RoboDK station: ClassTest.rdk

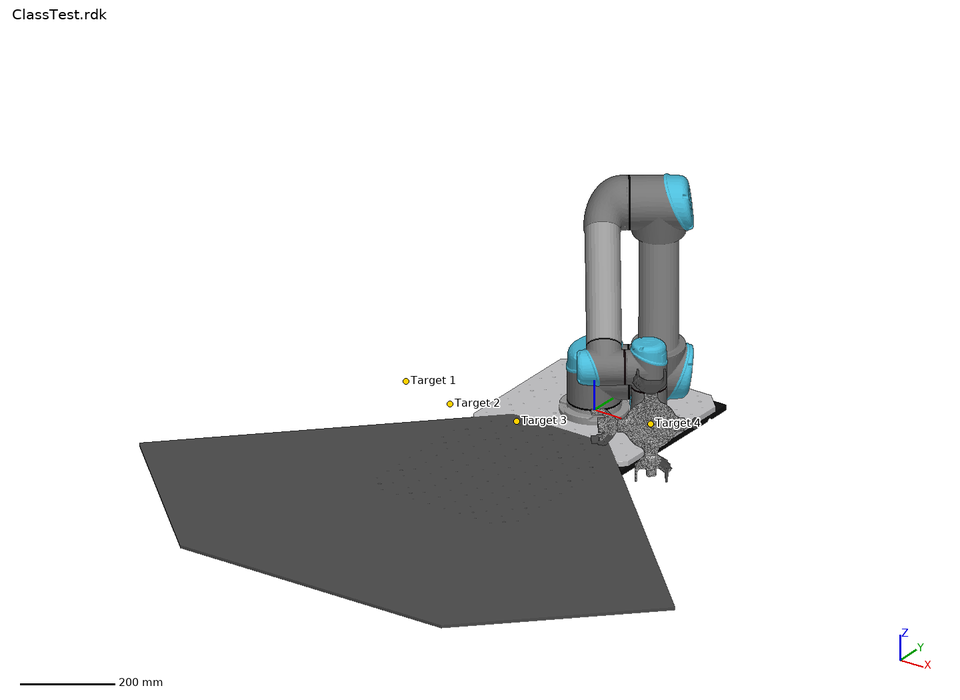
[picture v0: the station drawn from its stored meshes, robots at their saved joint values, targets as dots, program paths as lines]
Station P2 - Robot Cell (saved by RoboDK 5.5.3). Poses are relative to the parent item; angles as X-Y-Z fixed-axis rotations.
Station parameters (name, value as stored): IO_0, 0, IO_1, 1, 10, 0, 11, 0, 12, 1
  - frame UR5 Base at (0, 0, 0) mm
    - robot UR5: 6 axes
        modified DH rows (alpha deg, a mm, theta deg, d mm): 0, 0, 0, 89.2; 90, 0, 180, 0; 0, 425, 0, 0; 0, 392, 0, 109.3; -90, 0, 0, 94.75; 90, 0, 0, 82.5
        joint limits [-360, -360, -360, -360, -360, -360] to [360, 360, 360, 360, 360, 360]; home [0, -90, -90, 0, 90, 0]; saved at [125.87, -83.08, 119.4, -38.13, 88.09, -180]
      - tool GripperAssembled, TCP at (0, 0, 0) mm, size 226.2 x 248.1 x 43.3 mm, geometry from GripperAssembled.step
    - object RobotCellTable at (0, 0, 0) mm, rotated rx 0 ry 0 rz 180 deg, size 1378.2 x 1242.6 x 30 mm, geometry from RobotCellTable.step
    - target Target 1 (joint target) at (-183.8, -428.35, 186.83) mm, rotated rx 2.21 ry -88.19 rz 52.55 deg; joints [52.87, -83.08, 119.4, -38.13, 88.11, 89.99] of UR5
    - target Target 2 (joint target) at (-45.52, -463.89, 186.83) mm, rotated rx 88.19 ry 0.06 rz -17.62 deg; joints [70.49, -83.08, 119.4, -38.13, 88.11, 0] of UR5
    - target Target 3 (joint target) at (116.99, -451.2, 186.83) mm, rotated rx -1.89 ry 88.19 rz -89.37 deg; joints [90.63, -83.08, 119.4, -38.13, 88.11, -90] of UR5
    - target Target 4 (joint target) at (355.89, -301.01, 186.83) mm, rotated rx -88.19 ry -0.06 rz -142.24 deg; joints [125.87, -83.08, 119.4, -38.13, 88.11, -180] of UR5
    - target T5 (joint target) at (-183.78, -428.36, 186.83) mm, rotated rx -88.19 ry -0.06 rz 144.78 deg; joints [52.87, -83.08, 119.4, -38.13, 88.09, -180] of UR5
    - target T6 (joint target) at (-183.78, -428.36, 186.83) mm, rotated rx -88.19 ry -0.06 rz 144.78 deg; joints [54.36, -83.08, 119.4, -38.13, 88.09, -180] of UR5
    - target T7 (joint target) at (-183.78, -428.36, 186.83) mm, rotated rx -88.19 ry -0.06 rz 144.78 deg; joints [55.85, -83.08, 119.4, -38.13, 88.09, -180] of UR5
    - target T8 (joint target) at (-183.78, -428.36, 186.83) mm, rotated rx -88.19 ry -0.06 rz 144.78 deg; joints [57.339, -83.08, 119.4, -38.13, 88.09, -180] of UR5
    - target T9 (joint target) at (-183.78, -428.36, 186.83) mm, rotated rx -88.19 ry -0.06 rz 144.78 deg; joints [58.829, -83.08, 119.4, -38.13, 88.09, -180] of UR5
    - target T10 (joint target) at (-183.78, -428.36, 186.83) mm, rotated rx -88.19 ry -0.06 rz 144.78 deg; joints [60.319, -83.08, 119.4, -38.13, 88.09, -180] of UR5
    - target T11 (joint target) at (-183.78, -428.36, 186.83) mm, rotated rx -88.19 ry -0.06 rz 144.78 deg; joints [61.809, -83.08, 119.4, -38.13, 88.09, -180] of UR5
    - target T12 (joint target) at (-183.78, -428.36, 186.83) mm, rotated rx -88.19 ry -0.06 rz 144.78 deg; joints [63.299, -83.08, 119.4, -38.13, 88.09, -180] of UR5
    - target T13 (joint target) at (-183.78, -428.36, 186.83) mm, rotated rx -88.19 ry -0.06 rz 144.78 deg; joints [64.788, -83.08, 119.4, -38.13, 88.09, -180] of UR5
    - target T14 (joint target) at (-183.78, -428.36, 186.83) mm, rotated rx -88.19 ry -0.06 rz 144.78 deg; joints [66.278, -83.08, 119.4, -38.13, 88.09, -180] of UR5
    - target T15 (joint target) at (-183.78, -428.36, 186.83) mm, rotated rx -88.19 ry -0.06 rz 144.78 deg; joints [67.768, -83.08, 119.4, -38.13, 88.09, -180] of UR5
    - target T16 (joint target) at (-183.78, -428.36, 186.83) mm, rotated rx -88.19 ry -0.06 rz 144.78 deg; joints [69.258, -83.08, 119.4, -38.13, 88.09, -180] of UR5
    - target T17 (joint target) at (-183.78, -428.36, 186.83) mm, rotated rx -88.19 ry -0.06 rz 144.78 deg; joints [70.748, -83.08, 119.4, -38.13, 88.09, -180] of UR5
    - target T18 (joint target) at (-183.78, -428.36, 186.83) mm, rotated rx -88.19 ry -0.06 rz 144.78 deg; joints [72.237, -83.08, 119.4, -38.13, 88.09, -180] of UR5
    - target T19 (joint target) at (-183.78, -428.36, 186.83) mm, rotated rx -88.19 ry -0.06 rz 144.78 deg; joints [73.727, -83.08, 119.4, -38.13, 88.09, -180] of UR5
    - target T20 (joint target) at (-183.78, -428.36, 186.83) mm, rotated rx -88.19 ry -0.06 rz 144.78 deg; joints [75.217, -83.08, 119.4, -38.13, 88.09, -180] of UR5
    - target T21 (joint target) at (-183.78, -428.36, 186.83) mm, rotated rx -88.19 ry -0.06 rz 144.78 deg; joints [76.707, -83.08, 119.4, -38.13, 88.09, -180] of UR5
    - target T22 (joint target) at (-183.78, -428.36, 186.83) mm, rotated rx -88.19 ry -0.06 rz 144.78 deg; joints [78.197, -83.08, 119.4, -38.13, 88.09, -180] of UR5
    - target T23 (joint target) at (-183.78, -428.36, 186.83) mm, rotated rx -88.19 ry -0.06 rz 144.78 deg; joints [79.686, -83.08, 119.4, -38.13, 88.09, -180] of UR5
    - target T24 (joint target) at (-183.78, -428.36, 186.83) mm, rotated rx -88.19 ry -0.06 rz 144.78 deg; joints [81.176, -83.08, 119.4, -38.13, 88.09, -180] of UR5
    - target T25 (joint target) at (-183.78, -428.36, 186.83) mm, rotated rx -88.19 ry -0.06 rz 144.78 deg; joints [82.666, -83.08, 119.4, -38.13, 88.09, -180] of UR5
    - target T26 (joint target) at (-183.78, -428.36, 186.83) mm, rotated rx -88.19 ry -0.06 rz 144.78 deg; joints [84.156, -83.08, 119.4, -38.13, 88.09, -180] of UR5
    - target T27 (joint target) at (-183.78, -428.36, 186.83) mm, rotated rx -88.19 ry -0.06 rz 144.78 deg; joints [85.646, -83.08, 119.4, -38.13, 88.09, -180] of UR5
    - target T28 (joint target) at (-183.78, -428.36, 186.83) mm, rotated rx -88.19 ry -0.06 rz 144.78 deg; joints [87.135, -83.08, 119.4, -38.13, 88.09, -180] of UR5
    - target T29 (joint target) at (-183.78, -428.36, 186.83) mm, rotated rx -88.19 ry -0.06 rz 144.78 deg; joints [88.625, -83.08, 119.4, -38.13, 88.09, -180] of UR5
    - target T30 (joint target) at (-183.78, -428.36, 186.83) mm, rotated rx -88.19 ry -0.06 rz 144.78 deg; joints [90.115, -83.08, 119.4, -38.13, 88.09, -180] of UR5
    - target T31 (joint target) at (-183.78, -428.36, 186.83) mm, rotated rx -88.19 ry -0.06 rz 144.78 deg; joints [91.605, -83.08, 119.4, -38.13, 88.09, -180] of UR5
    - target T32 (joint target) at (-183.78, -428.36, 186.83) mm, rotated rx -88.19 ry -0.06 rz 144.78 deg; joints [93.094, -83.08, 119.4, -38.13, 88.09, -180] of UR5
    - target T33 (joint target) at (-183.78, -428.36, 186.83) mm, rotated rx -88.19 ry -0.06 rz 144.78 deg; joints [94.584, -83.08, 119.4, -38.13, 88.09, -180] of UR5
    - target T34 (joint target) at (-183.78, -428.36, 186.83) mm, rotated rx -88.19 ry -0.06 rz 144.78 deg; joints [96.074, -83.08, 119.4, -38.13, 88.09, -180] of UR5
    - target T35 (joint target) at (-183.78, -428.36, 186.83) mm, rotated rx -88.19 ry -0.06 rz 144.78 deg; joints [97.564, -83.08, 119.4, -38.13, 88.09, -180] of UR5
    - target T36 (joint target) at (-183.78, -428.36, 186.83) mm, rotated rx -88.19 ry -0.06 rz 144.78 deg; joints [99.054, -83.08, 119.4, -38.13, 88.09, -180] of UR5
    - target T37 (joint target) at (-183.78, -428.36, 186.83) mm, rotated rx -88.19 ry -0.06 rz 144.78 deg; joints [100.543, -83.08, 119.4, -38.13, 88.09, -180] of UR5
    - target T38 (joint target) at (-183.78, -428.36, 186.83) mm, rotated rx -88.19 ry -0.06 rz 144.78 deg; joints [102.033, -83.08, 119.4, -38.13, 88.09, -180] of UR5
    - target T39 (joint target) at (-183.78, -428.36, 186.83) mm, rotated rx -88.19 ry -0.06 rz 144.78 deg; joints [103.523, -83.08, 119.4, -38.13, 88.09, -180] of UR5
    - target T40 (joint target) at (-183.78, -428.36, 186.83) mm, rotated rx -88.19 ry -0.06 rz 144.78 deg; joints [105.013, -83.08, 119.4, -38.13, 88.09, -180] of UR5
    - target T41 (joint target) at (-183.78, -428.36, 186.83) mm, rotated rx -88.19 ry -0.06 rz 144.78 deg; joints [106.503, -83.08, 119.4, -38.13, 88.09, -180] of UR5
    - target T42 (joint target) at (-183.78, -428.36, 186.83) mm, rotated rx -88.19 ry -0.06 rz 144.78 deg; joints [107.992, -83.08, 119.4, -38.13, 88.09, -180] of UR5
    - target T43 (joint target) at (-183.78, -428.36, 186.83) mm, rotated rx -88.19 ry -0.06 rz 144.78 deg; joints [109.482, -83.08, 119.4, -38.13, 88.09, -180] of UR5
    - target T44 (joint target) at (-183.78, -428.36, 186.83) mm, rotated rx -88.19 ry -0.06 rz 144.78 deg; joints [110.972, -83.08, 119.4, -38.13, 88.09, -180] of UR5
    - target T45 (joint target) at (-183.78, -428.36, 186.83) mm, rotated rx -88.19 ry -0.06 rz 144.78 deg; joints [112.462, -83.08, 119.4, -38.13, 88.09, -180] of UR5
    - target T46 (joint target) at (-183.78, -428.36, 186.83) mm, rotated rx -88.19 ry -0.06 rz 144.78 deg; joints [113.952, -83.08, 119.4, -38.13, 88.09, -180] of UR5
    - target T47 (joint target) at (-183.78, -428.36, 186.83) mm, rotated rx -88.19 ry -0.06 rz 144.78 deg; joints [115.441, -83.08, 119.4, -38.13, 88.09, -180] of UR5
    - target T48 (joint target) at (-183.78, -428.36, 186.83) mm, rotated rx -88.19 ry -0.06 rz 144.78 deg; joints [116.931, -83.08, 119.4, -38.13, 88.09, -180] of UR5
    - target T49 (joint target) at (-183.78, -428.36, 186.83) mm, rotated rx -88.19 ry -0.06 rz 144.78 deg; joints [118.421, -83.08, 119.4, -38.13, 88.09, -180] of UR5
    - target T50 (joint target) at (-183.78, -428.36, 186.83) mm, rotated rx -88.19 ry -0.06 rz 144.78 deg; joints [119.911, -83.08, 119.4, -38.13, 88.09, -180] of UR5
    - target T51 (joint target) at (-183.78, -428.36, 186.83) mm, rotated rx -88.19 ry -0.06 rz 144.78 deg; joints [121.401, -83.08, 119.4, -38.13, 88.09, -180] of UR5
    - target T52 (joint target) at (-183.78, -428.36, 186.83) mm, rotated rx -88.19 ry -0.06 rz 144.78 deg; joints [122.89, -83.08, 119.4, -38.13, 88.09, -180] of UR5
    - target T53 (joint target) at (-183.78, -428.36, 186.83) mm, rotated rx -88.19 ry -0.06 rz 144.78 deg; joints [124.38, -83.08, 119.4, -38.13, 88.09, -180] of UR5
    - target T54 (joint target) at (-183.78, -428.36, 186.83) mm, rotated rx -88.19 ry -0.06 rz 144.78 deg; joints [125.87, -83.08, 119.4, -38.13, 88.09, -180] of UR5
  - Python program Prog2 (listed below)
  - program Test program (53 instructions, listed below)
  - program Prog3 (2 instructions, listed below)

--- Python program Prog2 ---
from robodk import robolink    # RoboDK API
from robodk import robomath    # Robot toolbox

RDK = robolink.Robolink()

# Notify user:
print('To edit this program:\nright click on the Python program, then, select "Edit Python script"')

robot = RDK.Item("UR5")
RDK.setRunMode(1)

target1 = RDK.Item("T7")
target2 = RDK.Item("T30")
target3 = RDK.Item("T48")

val1 = list(target1.Joints()[0])
val2 = list(target2.Joints()[0])
val3 = list(target3.Joints()[0])

done1 = False
done2 = False
done3 = False

robot.setDO(11, 0)
robot.setDO(12, 0)


# Program example:
while True:

    rob_pose = robot.Joints()

    if val1[0][0] >= val2[0][0] and not done1:
        RDK.ShowMessage("Turning on the topgripper")
        robot.setDO(11, 1)
        done1 = True
    elif val2[0][0] >= val2[0][0] and not done2:
        RDK.ShowMessage("Turning on the pcbgripper")
        robot.setDO(12, 1)
        done2 = True
    elif val3[0][0] >= val2[0][0] and not done3:
        RDK.ShowMessage("Turning on the botgripper")
        done3 = True
        robot.setDO(11, 0)
        break

--- program Test program (robot UR5) ---
  Set Ref.: UR5 Base
  Set Tool at (0, 0, 0) mm
  Smooth(1)
  Set speed (100.0 mm/s)
  MoveL (T6)
  MoveL (T7)
  MoveL (T8)
  MoveL (T9)
  MoveL (T10)
  MoveL (T11)
  MoveL (T12)
  MoveL (T13)
  MoveL (T14)
  MoveL (T15)
  MoveL (T16)
  MoveL (T17)
  MoveL (T18)
  MoveL (T19)
  MoveL (T20)
  MoveL (T21)
  MoveL (T22)
  MoveL (T23)
  MoveL (T24)
  MoveL (T25)
  MoveL (T26)
  MoveL (T27)
  MoveL (T28)
  MoveL (T29)
  MoveL (T30)
  MoveL (T31)
  MoveL (T32)
  MoveL (T33)
  MoveL (T34)
  MoveL (T35)
  MoveL (T36)
  MoveL (T37)
  MoveL (T38)
  MoveL (T39)
  MoveL (T40)
  MoveL (T41)
  MoveL (T42)
  MoveL (T43)
  MoveL (T44)
  MoveL (T45)
  MoveL (T46)
  MoveL (T47)
  MoveL (T48)
  MoveL (T49)
  MoveL (T50)
  MoveL (T51)
  MoveL (T52)
  MoveL (T53)
  MoveL (T54)

--- program Prog3 (robot UR5) ---
  Run Prog2
  Call Test program
